// TIA Portal V19 export
DATA_BLOCK "FU_In_Out"   // DB222
{ S7_Optimized_Access := 'FALSE' }
// stored: AutoNumber false
   VAR RETAIN
      Anzahl : Int := 7;   // * Anzahl der zu bedienenden FUs
      Offset : Int := 10;   // * Beginn Daten erster FU
      Leng : Int := 16;   // * Länge einer FU-Struktur
      Fehler_Quitt : Bool := TRUE;
      res1 : Bool := FALSE;
      res2 : Bool := FALSE;
      res3 : Bool := FALSE;
      res4 : Bool := FALSE;
      res5 : Bool := FALSE;
      res6 : Bool := FALSE;
      res7 : Bool := FALSE;
      resB : Byte := 16#00;
      akt_FU : Int := 0;   // Zähler für FU-Bearbeitung
      FU : Array[1..15] of Struct
         Adresse : Int;   // * Adresse EA
         Fehler : Bool;   // Fehlerstatus Altmerker
         res : Bool;
         res1 : Bool;
         res2 : Bool;
         res3 : Bool;
         res4 : Bool;
         res5 : Bool;
         res6 : Bool;
         AM_Fehlernummer : USInt;   // Altmerker Fehlernummer
         PE : Struct
            Statusbyte : Struct
               Fehlernummer : USInt;   // nur bei Stoerung/Warunung
               Endfrei : Bool;   // Freigabe Endstufe
               Bereit : Bool;   // FU betriebsbereit
               PA_Dat : Bool;   // PA Daten freigegeben
               Akt_Intsatz : Bool;   // aktueller Integratorsatz
               Akt_Parsatz : Bool;   // aktueller Parametersatz
               Stoer : Bool;   // Stoerung/Warnung
               End_rechts : Bool;   // Endschalter rechts aktiv
               End_links : Bool;   // Endschalter links aktiv
            END_STRUCT;
            Speed : Int;
            Reserve : Word;
         END_STRUCT;
         PA : Struct
            Steuerwort : Struct
               resB : Byte;
               RegSp : Bool;   // Reglersperre
               FrgStop : Bool;   // Freigabe/Schnellstop
               FrgHalt : Bool;   // Freigabe/Halt
               HaltRg : Bool;   // Haltregelung
               IntUms : Bool;   // Integrator-Umschaltung
               ParUms : Bool;   // Parametersatz-Umschaltung
               Reset : Bool;   // Reset
               res : Bool;
            END_STRUCT;
            Speed : Int;
            Reserve : Word;
         END_STRUCT;
      END_STRUCT;
   END_VAR
BEGIN
   FU[1].Adresse := 1010;
   FU[2].Adresse := 1020;
   FU[3].Adresse := 1030;
   FU[4].Adresse := 1040;
   FU[5].Adresse := 1050;
   FU[6].Adresse := 1060;
   FU[7].Adresse := 1070;
   FU[8].Adresse := 1080;
   FU[9].Adresse := 1090;
   FU[10].Adresse := 0;
   FU[1..10].Fehler := FALSE;
   FU[1..10].res := FALSE;
   FU[1..10].res1 := FALSE;
   FU[1..10].res2 := FALSE;
   FU[1..10].res3 := FALSE;
   FU[1..10].res4 := FALSE;
   FU[1..10].res5 := FALSE;
   FU[1..10].res6 := FALSE;
   FU[1..10].AM_Fehlernummer := 16#00;
   FU[1..10].PE.Statusbyte.Fehlernummer := 16#00;
   FU[1..10].PE.Statusbyte.Endfrei := FALSE;
   FU[1..10].PE.Statusbyte.Bereit := FALSE;
   FU[1..10].PE.Statusbyte.PA_Dat := FALSE;
   FU[1..10].PE.Statusbyte.Akt_Intsatz := FALSE;
   FU[1..10].PE.Statusbyte.Akt_Parsatz := FALSE;
   FU[1..10].PE.Statusbyte.Stoer := FALSE;
   FU[1..10].PE.Statusbyte.End_rechts := FALSE;
   FU[1..10].PE.Statusbyte.End_links := FALSE;
   FU[1..5].PE.Speed := 0;
   FU[6].PE.Speed := 6750;
   FU[7..10].PE.Speed := 0;
   FU[1..10].PE.Reserve := 16#0000;
   FU[1..10].PA.Steuerwort.resB := 16#00;
   FU[1..4].PA.Steuerwort.RegSp := FALSE;
   FU[5].PA.Steuerwort.RegSp := TRUE;
   FU[6].PA.Steuerwort.RegSp := FALSE;
   FU[7..9].PA.Steuerwort.RegSp := TRUE;
   FU[10].PA.Steuerwort.RegSp := FALSE;
   FU[1..5].PA.Steuerwort.FrgStop := FALSE;
   FU[6].PA.Steuerwort.FrgStop := TRUE;
   FU[7..10].PA.Steuerwort.FrgStop := FALSE;
   FU[1..5].PA.Steuerwort.FrgHalt := FALSE;
   FU[6].PA.Steuerwort.FrgHalt := TRUE;
   FU[7..10].PA.Steuerwort.FrgHalt := FALSE;
   FU[1..10].PA.Steuerwort.HaltRg := FALSE;
   FU[1..10].PA.Steuerwort.IntUms := FALSE;
   FU[1..10].PA.Steuerwort.ParUms := FALSE;
   FU[1..10].PA.Steuerwort.Reset := FALSE;
   FU[1..10].PA.Steuerwort.res := FALSE;
   FU[1..5].PA.Speed := 0;
   FU[6].PA.Speed := 6750;
   FU[7..10].PA.Speed := 0;
   FU[1..10].PA.Reserve := 16#0000;
END_DATA_BLOCK
